Fanuc KAREL source: kb00069.KL

-- PROVISIONAL review KL for V940-1; original PC SHA256 e7907af303c44355d021b95c613ef27cab1d8ceef76a68fec6bf2faddefe0a57
-- Incomplete behavior may be omitted. Consult companion uncertainty JSON. Do not deploy.
PROGRAM KB00069
%NOLOCKGROUP
BEGIN
  -- V9_ZERO_TABLE_METADATA_HINT layout=0002_ascii; no indexed target words; source/name/runtime held
  -- UNRESOLVED_PC offsets 5-14; opcodes 3F,75
  -- UNRESOLVED_PC offsets 19-26; opcodes 9D,23
  -- UNRESOLVED_PC offsets 31-40; opcodes 3F,75
  -- UNRESOLVED_PC offsets 45-52; opcodes 9D,23
  -- UNRESOLVED_PC offsets 57-89; opcodes 27,22,2A,22,22,2A,22,31
  -- UNRESOLVED_PC offsets 94-98; opcodes 7F
END KB00069
